FUNCTION PoundsPerSquareInchToPascal : Pascal
VAR_INPUT
    pressure : PoundsPerSquareInch;
END_VAR

PoundsPerSquareInchToPascal._ := pressure._ * 6895;

END_FUNCTION

(* stored: Version 1.1.0.1, ProductVersion 3.1.4024.4
   POU PoundsPerSquareInchToPascal: Id {a948ff2b-09b1-41f7-99ac-1d3332b14541}, SpecialFunc None *)
